// Mitsubishi GX Works2 project: robot   PLC: Q03UDV

PROGRAM MAIN
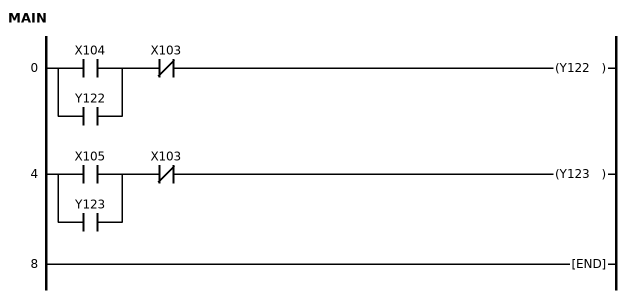
0     LD      X104
      OR      Y122
      ANI     X103
      OUT     Y122
4     LD      X105
      OR      Y123
      ANI     X103
      OUT     Y123
8     END
END_PROGRAM
